// TIA Portal V20 export
// export: Created 2025-09-12T17:59:00.0000000Z, ExportSetting WithDefaults
FUNCTION_BLOCK "FB500_EM_Monitoring"   // FB, SCL
TITLE = EM-500: System Monitoring
AUTHOR : Dallas Levine
VERSION : 0.1
// This block contains all logic for the Monitoring Equipment Module (EM-500).
// stored: AutoNumber true, IsRetain false
   VAR_INPUT
      Enable : Bool;   // Enables the block's execution.
   END_VAR
   VAR
      UDT : "UDT500_EM_Monitoring";   // The data interface for the Monitoring Equipment Module.
   END_VAR
BEGIN
   REGION Placeholder for SCL Code 

   END_REGION
END_FUNCTION_BLOCK
